// TIA Portal V16 export
// export: Created 2023-09-11T12:14:51.705076Z, ExportSetting WithDefaults, DisplayName Totally Integrated Automation Portal, DisplayVersion V16 Update 6, DisplayName TIA Portal Version Control Interface, DisplayVersion V16 Update 2, DisplayName TIA Portal Openness, DisplayVersion V16 Update 6, DisplayName STEP 7 Professional, DisplayVersion V16 Update 6, DisplayName STEP 7 Safety, DisplayVersion V16, DisplayName WinCC Advanced, DisplayVersion V16 Update 6
FUNCTION_BLOCK "01_E_Inverter current overload control"   // FB17, LAD
TITLE = Control Current Overload
{ S7_Optimized_Access := 'TRUE' }
AUTHOR : rtecmer
VERSION : 0.1
// Kontrola przeciążenia invertera KDN M25 M27
// stored: AutoNumber true, IsIECCheckEnabled false, IsRetainMemResEnabled false, MemoryReserve 500, SetENOAutomatically false, UDAEnableTagReadback false
BEGIN

REGION Network 1: Ustawienie wartości granicznej
   // Nastawa dopuszczalnego prądu invertera. Znacznik M10 zastosowany w celach serwisowych. Wybór ograniczenia z edytowanego z HMI lub z nastaw czytanych z falownika.
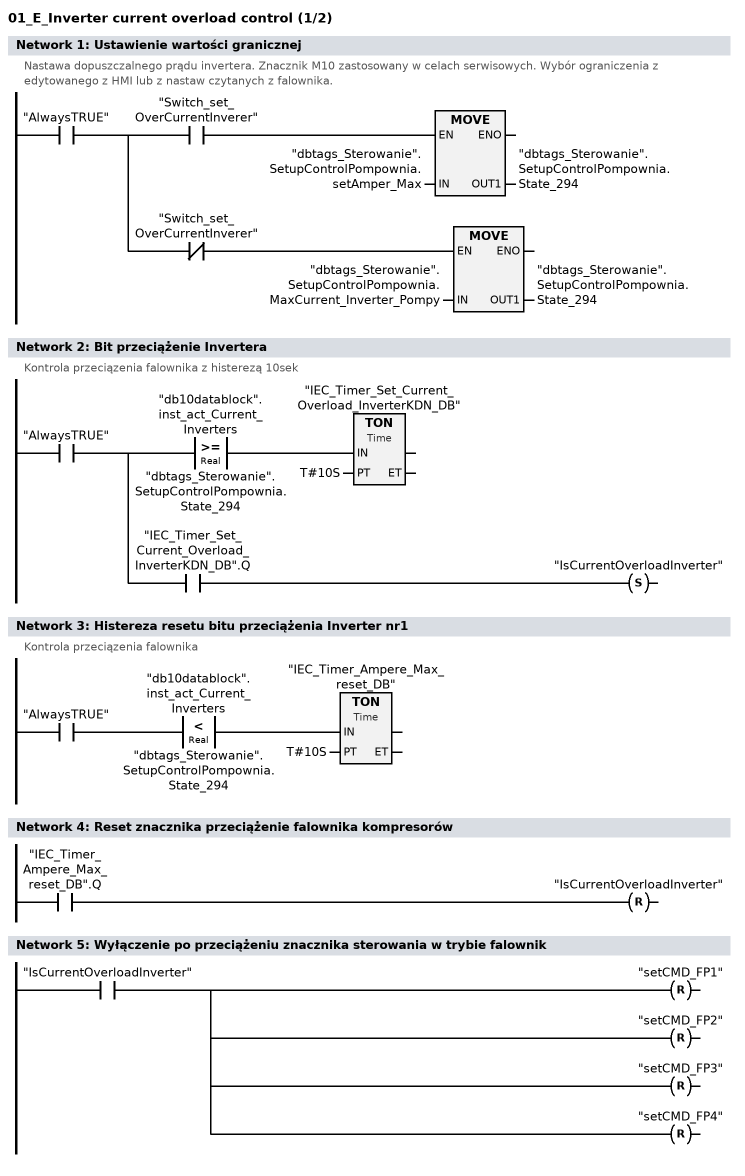
   RUNG wire#powerrail
      Contact( "AlwaysTRUE" )
      wire#w1
      Contact( "Switch_set_OverCurrentInverer" )
      Move(in := "dbtags_Sterowanie".SetupControlPompownia.setAmper_Max, out1 => "dbtags_Sterowanie".SetupControlPompownia.State_294)
   END_RUNG
   RUNG wire#w1
      I_Contact( "Switch_set_OverCurrentInverer" )
      Move(in := "dbtags_Sterowanie".SetupControlPompownia.MaxCurrent_Inverter_Pompy, out1 => "dbtags_Sterowanie".SetupControlPompownia.State_294)
   END_RUNG
   // the same network as SCL:
   IF "AlwaysTRUE" AND "Switch_set_OverCurrentInverer" THEN
       "dbtags_Sterowanie".SetupControlPompownia.State_294 := "dbtags_Sterowanie".SetupControlPompownia.setAmper_Max;
   END_IF;
   IF "AlwaysTRUE" AND NOT "Switch_set_OverCurrentInverer" THEN
       "dbtags_Sterowanie".SetupControlPompownia.State_294 := "dbtags_Sterowanie".SetupControlPompownia.MaxCurrent_Inverter_Pompy;
   END_IF;
END_REGION

REGION Network 2: Bit przeciążenie Invertera
   // Kontrola przeciązenia falownika z histerezą 10sek
   RUNG wire#powerrail
      Contact( "AlwaysTRUE" )
      wire#w1
      { S7_Templates := "SrcType := Real" } GE_Contact(in1 := "db10datablock".inst_act_Current_Inverters, in2 := "dbtags_Sterowanie".SetupControlPompownia.State_294)
      { S7_Templates := "time_type := Time" } "IEC_Timer_Set_Current_Overload_InverterKDN_DB".TON(pt := T#10S, et =>)
   END_RUNG
   RUNG wire#w1
      Contact( "IEC_Timer_Set_Current_Overload_InverterKDN_DB".Q )
      S_Coil( "IsCurrentOverloadInverter" )
   END_RUNG
   // the same network as SCL:
   "IEC_Timer_Set_Current_Overload_InverterKDN_DB".TON(IN := "AlwaysTRUE" AND ("db10datablock".inst_act_Current_Inverters >= "dbtags_Sterowanie".SetupControlPompownia.State_294),
                           PT := T#10S);
   IF "AlwaysTRUE" AND "IEC_Timer_Set_Current_Overload_InverterKDN_DB".Q THEN
       "IsCurrentOverloadInverter" := TRUE;
   END_IF;
END_REGION

REGION Network 3: Histereza resetu bitu przeciążenia Inverter nr1
   // Kontrola przeciązenia falownika
   RUNG wire#powerrail
      Contact( "AlwaysTRUE" )
      { S7_Templates := "SrcType := Real" } LT_Contact(in1 := "db10datablock".inst_act_Current_Inverters, in2 := "dbtags_Sterowanie".SetupControlPompownia.State_294)
      { S7_Templates := "time_type := Time" } "IEC_Timer_Ampere_Max_reset_DB".TON(pt := T#10S, et =>)
   END_RUNG
   // the same network as SCL:
   "IEC_Timer_Ampere_Max_reset_DB".TON(IN := "AlwaysTRUE" AND ("db10datablock".inst_act_Current_Inverters < "dbtags_Sterowanie".SetupControlPompownia.State_294),
                           PT := T#10S);
END_REGION

REGION Network 4: Reset znacznika przeciążenie falownika kompresorów
   RUNG wire#powerrail
      Contact( "IEC_Timer_Ampere_Max_reset_DB".Q )
      R_Coil( "IsCurrentOverloadInverter" )
   END_RUNG
   // the same network as SCL:
   IF "IEC_Timer_Ampere_Max_reset_DB".Q THEN "IsCurrentOverloadInverter" := FALSE; END_IF;
END_REGION

REGION Network 5: Wyłączenie po przeciążeniu znacznika sterowania w trybie falownik
   RUNG wire#powerrail
      Contact( "IsCurrentOverloadInverter" )
      wire#w1
      R_Coil( "setCMD_FP1" )
   END_RUNG
   RUNG wire#w1
      R_Coil( "setCMD_FP2" )
   END_RUNG
   RUNG wire#w1
      R_Coil( "setCMD_FP3" )
   END_RUNG
   RUNG wire#w1
      R_Coil( "setCMD_FP4" )
   END_RUNG
   // the same network as SCL:
   IF "IsCurrentOverloadInverter" THEN
       "setCMD_FP1" := FALSE;
       "setCMD_FP2" := FALSE;
       "setCMD_FP3" := FALSE;
       "setCMD_FP4" := FALSE;
   END_IF;
END_REGION

REGION Network 6: Wyłączenie po przeciążeniu znacznika sterowania w trybie falownik
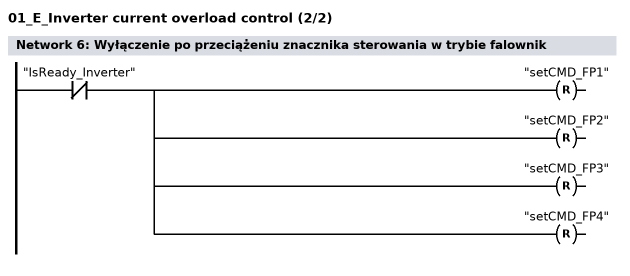
   RUNG wire#powerrail
      I_Contact( "IsReady_Inverter" )
      wire#w1
      R_Coil( "setCMD_FP1" )
   END_RUNG
   RUNG wire#w1
      R_Coil( "setCMD_FP2" )
   END_RUNG
   RUNG wire#w1
      R_Coil( "setCMD_FP3" )
   END_RUNG
   RUNG wire#w1
      R_Coil( "setCMD_FP4" )
   END_RUNG
   // the same network as SCL:
   IF NOT "IsReady_Inverter" THEN
       "setCMD_FP1" := FALSE;
       "setCMD_FP2" := FALSE;
       "setCMD_FP3" := FALSE;
       "setCMD_FP4" := FALSE;
   END_IF;
END_REGION
END_FUNCTION_BLOCK
